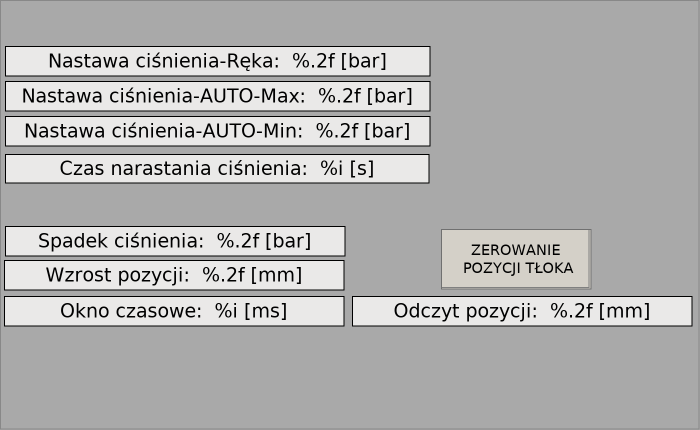
VISUALIZATION E2  // 700x430
    Textfield (5,81 425x30), "Nastawa ciśnienia-AUTO-Max: %.2f [bar]", text variable: GVL_HMI.PressureSetpointAutoMax
        OnMouseDown: write the text variable via Default, min 0, max 300
    Textfield (5,46 425x30), "Nastawa ciśnienia-Ręka: %.2f [bar]", text variable: GVL_HMI.nPressureSetpointManual
        OnMouseDown: write the text variable via Default, min 0, max 200
    Textfield (5,116 425x30), "Nastawa ciśnienia-AUTO-Min: %.2f [bar]", text variable: GVL_HMI.PressureSetpointAutoMin
        OnMouseDown: write the text variable via Default, min 0, max 300
    Textfield (5,226 340x30), "Spadek ciśnienia: %.2f [bar]", text variable: GVL_HMI.nBreakDeltaPress
        OnMouseDown: write the text variable via Default, min 0, max 200
    Textfield (4,260 340x30), "Wzrost pozycji: %.2f [mm]", text variable: GVL_HMI.nBreakDeltaPos
        OnMouseDown: write the text variable via Default, min 0, max 200
    Textfield (4,296 340x30), "Okno czasowe: %i [ms]", text variable: GVL_HMI.nBreak_Time_Window
        OnMouseDown: write the text variable via Default, min 0, max 200
    Textfield (5,154 424x29), "Czas narastania ciśnienia: %i [s]", text variable: GVL_HMI.nRamp_Time
        OnMouseDown: write the text variable via Default, min 0, max 3600
    Textfield (352,296 340x30), "Odczyt pozycji: %.2f [mm]", text variable: Scaling.fbPos.PosZeroed_mm
    Button (441,229 150x60), "ZEROWANIE POZYCJI TŁOKA", input disabled if: bLedCycleOn
        OnMouseDown: execute { Scaling.fbPos.SetZero:=false; }
        OnMouseUp: execute { Scaling.fbPos.SetZero:=true; }
END_VISUALIZATION

(* stored: Version 1.1.0.1, ProductVersion 3.1.4024.16
   Visu E2: Id {4a084321-3052-49a3-bb93-02bc66fb0e92} *)
